{region '#Template'}
	{attribute 'Category' := 'Universal'}
	{attribute 'Version' := '0.0.1.0'}
	{attribute 'Tags' := 'Universal, Control, PID, Loop'}
	{attribute 'Description' := 'Regler	// Controller'}
{endregion}
FUNCTION_BLOCK FB_BA_PID_Sp EXTENDS FB_BA_View
VAR_INPUT
	bEn						: BOOL;
	fX						: REAL;
	bSync					: BOOL;
	fSync					: REAL;
END_VAR
VAR_OUTPUT
	fY						: REAL;
	fMax					: REAL;
	fMin					: REAL;	
END_VAR
VAR_INPUT CONSTANT
	Sp						: FB_BA_AV_Op;		 
	Ctrl					: FB_BA_Loop;	
END_VAR

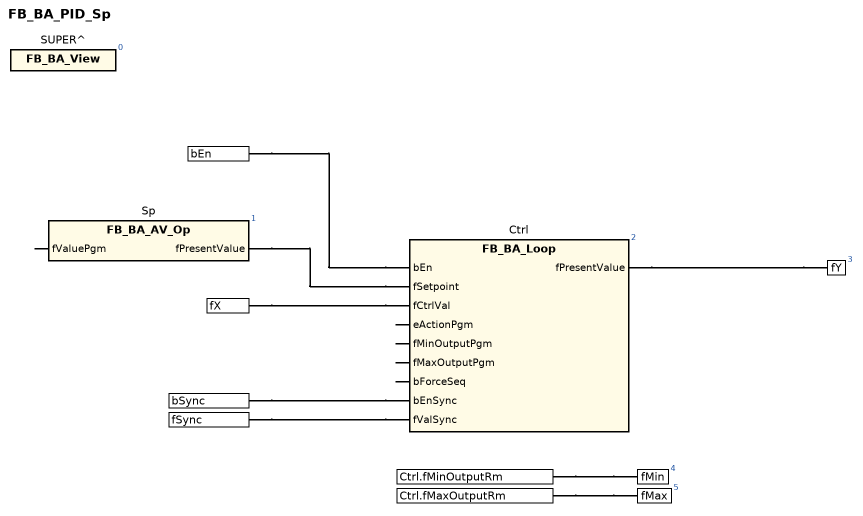
SUPER^(); // FB_BA_View
Sp(); // FB_BA_AV_Op
Ctrl(bEn := bEn, fSetpoint := Sp.fPresentValue, fCtrlVal := fX, bEnSync := bSync, fValSync := fSync); // FB_BA_Loop
fY := Ctrl.fPresentValue;
fMin := Ctrl.fMinOutputRm;
fMax := Ctrl.fMaxOutputRm;

METHOD FB_init : BOOL
VAR_INPUT
	bInitRetains : BOOL; // if TRUE, the retain variables are initialized (warm start / cold start)
	bInCopyCode : BOOL;  // if TRUE, the instance afterwards gets moved into the copy code (online change)
END_VAR
Sp.iParent					:= THIS^;
Sp.iLabel					:= LblUniControl.PID_Sp;		 
Sp.sObjectName				:= '{Idx=01}';								 	 
Sp.eUnit 					:= E_BA_Unit.eTemperature_DegreesCelsius;								 
Sp.fValueRm					:= 21.0;															 
Sp.fCOVIncrement			:= BA2_Param.fDefCOVIncrement;

Ctrl.iParent				:= THIS^;
Ctrl.iLabel					:= LblUniControl.PID_Ctrl; 
Ctrl.sObjectName			:= '{Idx=01}';
Ctrl.eOpMode				:= BA2_Param.nLoop_DefOpMode;								 	 										 
Ctrl.eOutputUnit			:= E_BA_Unit.eOther_Percent;
Ctrl.eActionRm				:= E_BA_Action.eReverse;
Ctrl.fProportionalConstant	:= 3;
Ctrl.fIntegralConstant		:= 180;
Ctrl.fDerivativeConstant	:= 0;
Ctrl.fMaxOutputRm 			:= 100;
Ctrl.fMinOutputRm			:= 0;
Ctrl.fCOVIncrement			:= 0;
Ctrl.nDampConstant			:= 0;
Ctrl.fNeutralZone			:= 0;
Ctrl.stStepDelay.nDown		:= 0;
Ctrl.stStepDelay.nUp		:= 0;
END_METHOD

END_FUNCTION_BLOCK

(* stored: Version 1.1.0.1, ProductVersion 3.1.4024.6
   POU FB_BA_PID_Sp: Id {780dc846-72bd-4d57-9166-e6f48cd6c151}, SpecialFunc None
   Method FB_init: Id {3386f0f2-178d-4227-a45d-7737d5736a7c} *)
